FUNCTION_BLOCK FB_Building
VAR_INPUT
END_VAR
VAR_OUTPUT
END_VAR
VAR
	_aFloors	: ARRAY [1..5] OF FB_Floor;
END_VAR

METHOD CalcPowerConsumption : UDINT
VAR
	nFloor		: INT;
END_VAR
FOR nFloor := 1 TO 5 DO
	CalcPowerConsumption := CalcPowerConsumption + refFloors[nFloor].CalcPowerConsumption();
END_FOR
END_METHOD

PROPERTY refFloors : REFERENCE TO ARRAY [1..5] OF FB_Floor
GET
refFloors REF= THIS^._aFloors;
END_GET
END_PROPERTY

END_FUNCTION_BLOCK

(* stored: Version 1.1.0.1, ProductVersion 3.1.4024.12
   POU FB_Building: Id {89a8e256-b6ab-4c49-bfea-2876b915c770}, SpecialFunc None
   Method CalcPowerConsumption: Id {03b69ec9-fecf-4cbb-bb31-8281e8ec4216}
   Property refFloors: Id {dd468346-9fa3-45b8-8f7d-931775cd8222}
   Get Get: Id {9d190e2d-51c7-47e5-84d9-546f7e5f3241} *)
